(* PLC project momentary_button, Dassault Systèmes ControlBuild 2024x *)
(* stored: creationDateTime 2023-10-03T11:13:21-01:00 *)

(* This module simulates a momentary contact push button. *)
FUNCTION_BLOCK equipment_library.momentary_button
  VAR_OUTPUT
    PB : BOOL := false;
  END_VAR
  VAR
    action : BOOL := false;
    timeCounter : REAL := 0.0;
  END_VAR
  VAR CONSTANT
    pulseDuration : REAL := 5.0;
    PBLogic : BOOL := true;
  END_VAR

(* -----------------------------------------------------------------	*)
(* Type : Model of Operative Behaviour					*)
(* Category :  Power								*)
(* Author : Dassault Systemes						*)
(* Update date : June 2018							*)
(* -----------------------------------------------------------------	*)
(* This module simulates a momentary contact push button. 		*)
(* -----------------------------------------------------------------	*)

IF (action) THEN
	timeCounter := timeCounter + ( CLOCK_PERIOD / 1000000.0);
	IF (timeCounter > pulseDuration) THEN
		action := FALSE;
		timeCounter := 0.0;
	END_IF;
END_IF;
PB := (action XOR NOT PBLogic);
END_FUNCTION_BLOCK
